FUNCTION_BLOCK Auto_rock
VAR_INPUT
	Safety_interlock:BOOL;
	Lh_depth:REAL;
	Rh_depth:REAL;
	Underground_despatch:BOOL;
	Right_brakes_on_dist:REAL;
	Left_brakes_on_dist:REAL;
	Tip_zone_up:REAL;
	Tip_zone_down:REAL;
	Box_zone_up:REAL;
	Box_zone_down:REAL;
	Rock_cycle_unlatch_dist:REAL;
	Loaded_skip_current:REAL;
END_VAR
VAR_OUTPUT
	Auto_ref:REAL;
	Starting_torque:REAL;
	Manual:BOOL;
	Auto:BOOL;
	Auto_go:BOOL;
	Auto_fwd:BOOL;
	Auto_rev:BOOL;
	Trail_brakes:BOOL;
	Fwd_incomplete:BOOL;
	Rev_incomplete:BOOL;
	Left_tip_zone:BOOL;
	Right_tip_zone:BOOL;
	Left_box_zone:BOOL;
	Right_box_zone:BOOL;
	Ready_to_load_rock:BOOL;
	Left_bank_zone:BOOL;
	Right_bank_zone:BOOL;
	ct_Skip_still_full:BOOL;
	ct_Auto_requirements:BOOL;
END_VAR
VAR_IN_OUT
	HMI_data:dut_Auto_rock;
	Levels:ARRAY[*] OF REAL;
END_VAR
VAR
	Auto_requirements_fault:BOOL;
	Rock_cycle_bypass_hmi:BOOL;
	Window_0: Window;
	Window_1: Window;
	R_TRIG_0: R_TRIG;
	R_TRIG_1: R_TRIG;
	TOF_0: TOF;
	F_TRIG_0: F_TRIG;
	BIT_TO_WORD_V0_0: BIT_TO_WORD_V0;
	WORD_TO_BIT_V0_0: WORD_TO_BIT_V0;
END_VAR

Zones();
Auto_mode();
Despatch();
Trail_brakes_m();
Auto_trips();
HMI_data_m();

METHOD Auto_mode
VAR_INPUT
END_VAR
VAR_INST // added by the converter: edge detectors and wires of the graphical bodies
    _w1, _w2 : BOOL;
    _w3 : ANY;
END_VAR
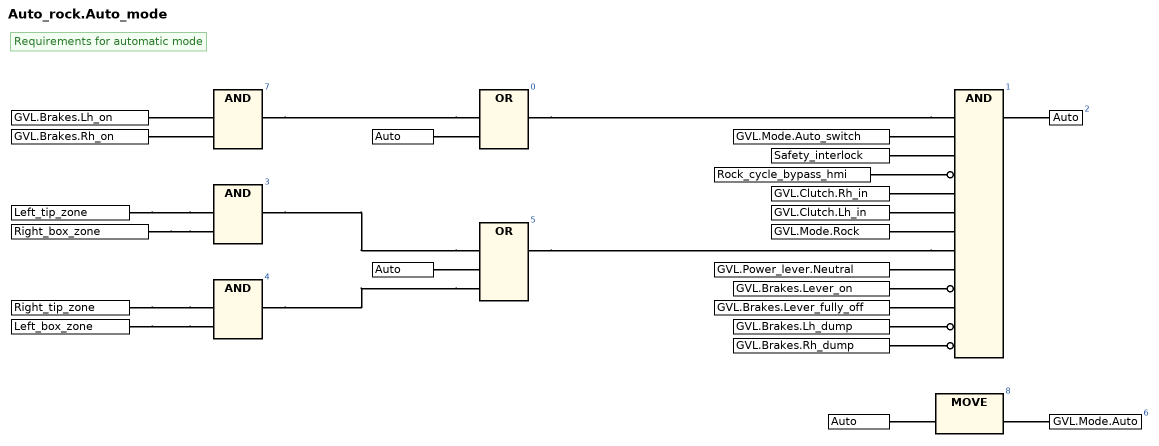
Auto := (_w1 OR Auto) AND GVL.Mode.Auto_switch AND Safety_interlock AND NOT Rock_cycle_bypass_hmi AND GVL.Clutch.Rh_in AND GVL.Clutch.Lh_in AND GVL.Mode.Rock AND _w2 AND GVL.Power_lever.Neutral AND NOT GVL.Brakes.Lever_on AND GVL.Brakes.Lever_fully_off AND NOT GVL.Brakes.Lh_dump AND NOT GVL.Brakes.Rh_dump;
_w2 := Left_tip_zone AND Right_box_zone OR Auto OR Right_tip_zone AND Left_box_zone;
GVL.Mode.Auto := _w3;
// Requirements for automatic mode
_w1 := GVL.Brakes.Lh_on AND GVL.Brakes.Rh_on;
_w3 := Auto;
END_METHOD

METHOD Auto_trips
VAR_INPUT
END_VAR
VAR_INST // added by the converter: edge detectors and wires of the graphical bodies
    _w1, _w2, _w3, _w4 : BOOL;
    _w5 : ANY;
END_VAR
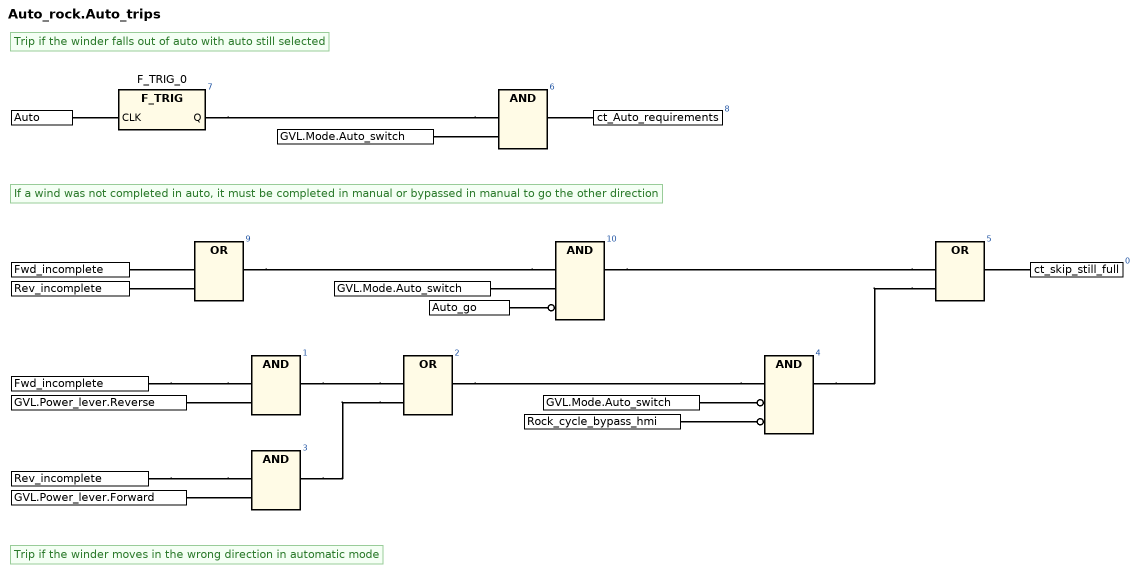
ct_skip_still_full := _w1;
_w3 := Fwd_incomplete AND GVL.Power_lever.Reverse OR _w2;
// Trip if the winder moves in the wrong direction in automatic mode
_w2 := Rev_incomplete AND GVL.Power_lever.Forward;
_w1 := _w4 OR _w3 AND NOT GVL.Mode.Auto_switch AND NOT Rock_cycle_bypass_hmi;
_w5 := F_TRIG_0.Q AND GVL.Mode.Auto_switch;
// Trip if the winder falls out of auto with auto still selected
F_TRIG_0(CLK := Auto); // F_TRIG
ct_Auto_requirements := _w5;
// If a wind was not completed in auto, it must be completed in manual or bypassed in manual to go the other direction
_w4 := (Fwd_incomplete OR Rev_incomplete) AND GVL.Mode.Auto_switch AND NOT Auto_go;
END_METHOD

METHOD Despatch
VAR_INPUT
END_VAR
VAR_INST // added by the converter: edge detectors and wires of the graphical bodies
    _w1, _w2, _w3, _w4, _w5, _w6, _w7, _w8, _w11, _w12, _w13 : BOOL;
    _w9, _w10 : REAL;
END_VAR
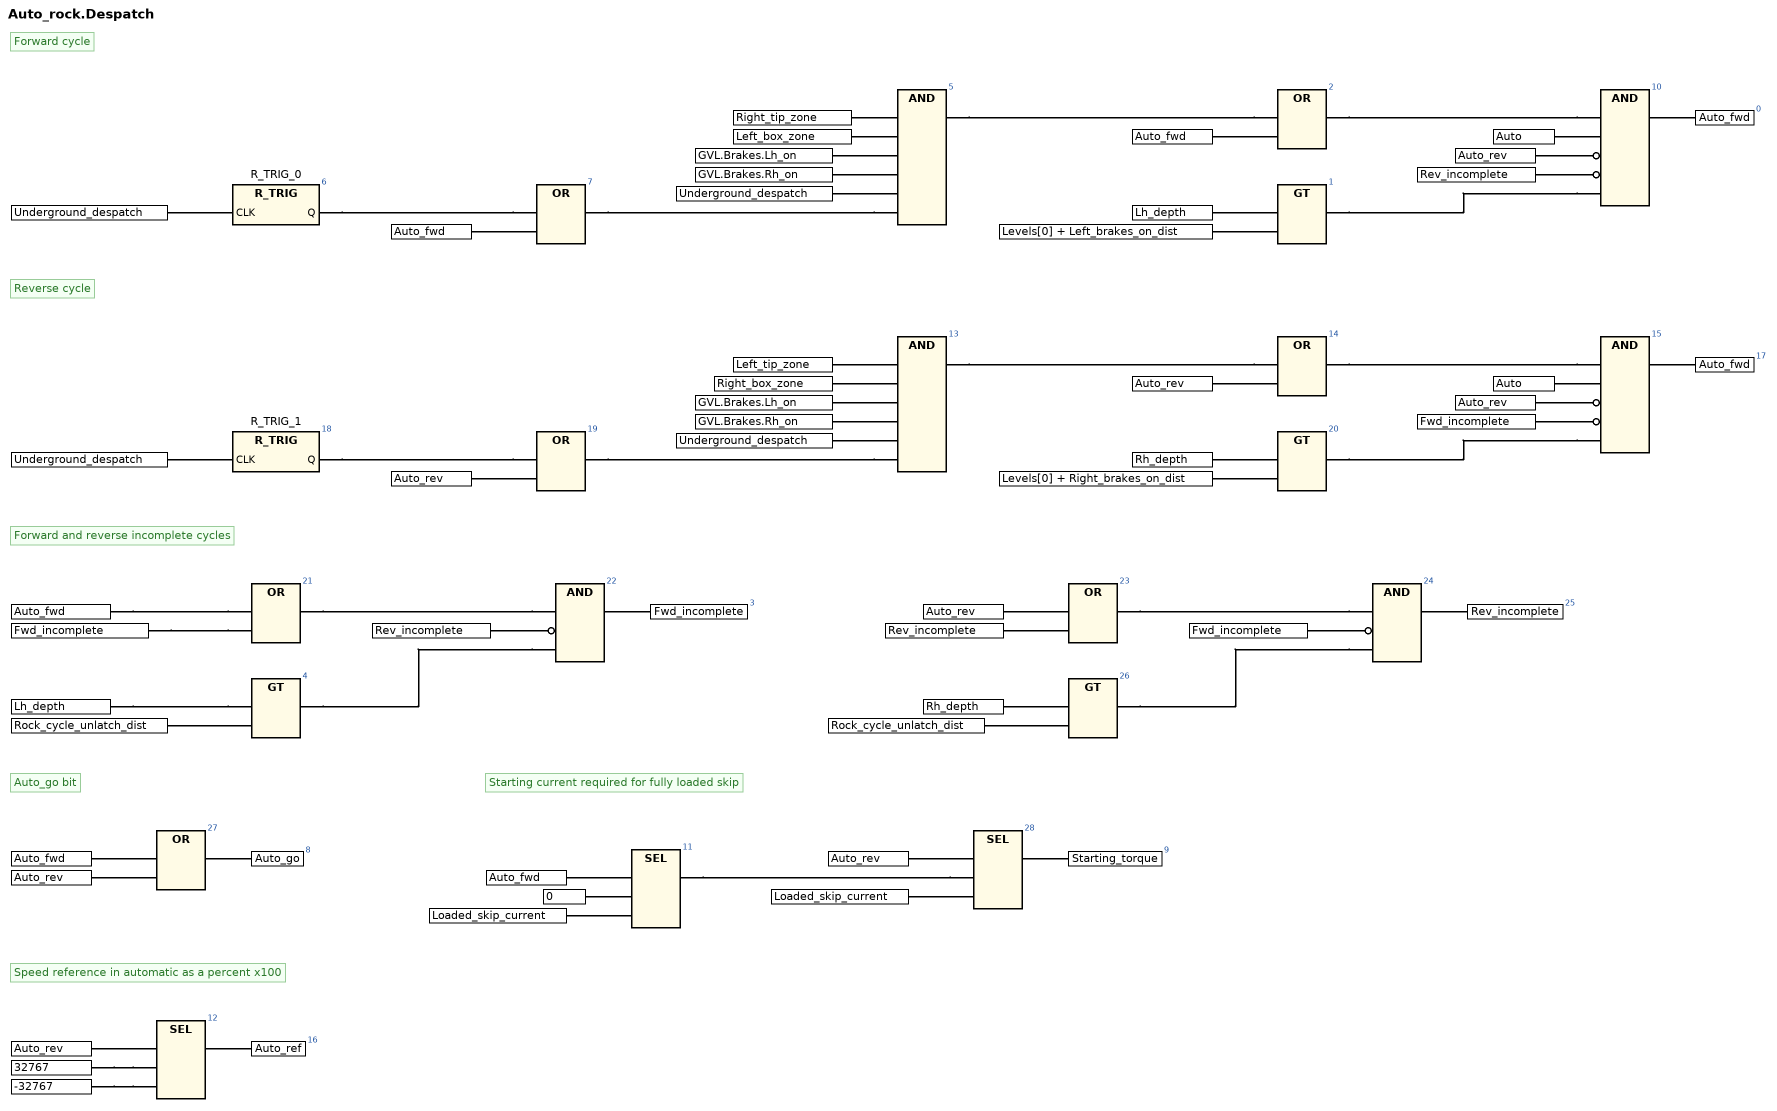
Auto_fwd := _w1;
_w2 := Lh_depth > (Levels[0] + Left_brakes_on_dist);
_w4 := _w3 OR Auto_fwd;
Fwd_incomplete := _w5;
_w6 := Lh_depth > Rock_cycle_unlatch_dist;
_w3 := Right_tip_zone AND Left_box_zone AND GVL.Brakes.Lh_on AND GVL.Brakes.Rh_on AND Underground_despatch AND _w7;
// Forward cycle
R_TRIG_0(CLK := Underground_despatch); // R_TRIG
_w7 := R_TRIG_0.Q OR Auto_fwd;
Auto_go := _w8;
Starting_torque := _w9;
_w1 := _w4 AND Auto AND NOT Auto_rev AND NOT Rev_incomplete AND _w2;
// Starting current required for fully loaded skip
_w10 := SEL(Auto_fwd, 0, Loaded_skip_current);
// Speed reference in automatic as a percent x100
Auto_ref := SEL(Auto_rev, 32767, -32767);
Auto_fwd := (Left_tip_zone AND Right_box_zone AND GVL.Brakes.Lh_on AND GVL.Brakes.Rh_on AND Underground_despatch AND _w11 OR Auto_rev) AND Auto AND NOT Auto_rev AND NOT Fwd_incomplete AND _w12;
// Reverse cycle
R_TRIG_1(CLK := Underground_despatch); // R_TRIG
_w11 := R_TRIG_1.Q OR Auto_rev;
_w12 := Rh_depth > (Levels[0] + Right_brakes_on_dist);
// Forward and reverse incomplete cycles
_w5 := (Auto_fwd OR Fwd_incomplete) AND NOT Rev_incomplete AND _w6;
Rev_incomplete := (Auto_rev OR Rev_incomplete) AND NOT Fwd_incomplete AND _w13;
_w13 := Rh_depth > Rock_cycle_unlatch_dist;
// Auto_go bit
_w8 := Auto_fwd OR Auto_rev;
_w9 := SEL(Auto_rev, _w10, Loaded_skip_current);
END_METHOD

METHOD HMI_data_m
VAR_INPUT
END_VAR
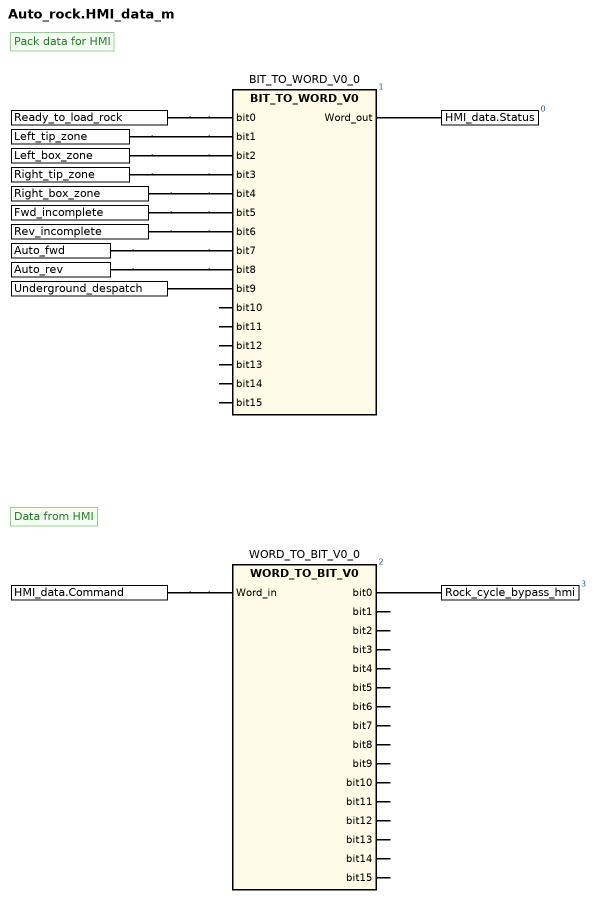
HMI_data.Status := BIT_TO_WORD_V0_0.Word_out;
// Pack data for HMI
BIT_TO_WORD_V0_0(
    bit0 := Ready_to_load_rock,
    bit1 := Left_tip_zone,
    bit2 := Left_box_zone,
    bit3 := Right_tip_zone,
    bit4 := Right_box_zone,
    bit5 := Fwd_incomplete,
    bit6 := Rev_incomplete,
    bit7 := Auto_fwd,
    bit8 := Auto_rev,
    bit9 := Underground_despatch); // BIT_TO_WORD_V0
// Data from HMI
WORD_TO_BIT_V0_0(Word_in := HMI_data.Command); // WORD_TO_BIT_V0
Rock_cycle_bypass_hmi := WORD_TO_BIT_V0_0.bit0;
END_METHOD

METHOD Trail_brakes_m
VAR_INPUT
END_VAR
VAR_INST // added by the converter: edge detectors and wires of the graphical bodies
    _w1, _w3 : BOOL;
    _w2 : ANY;
END_VAR
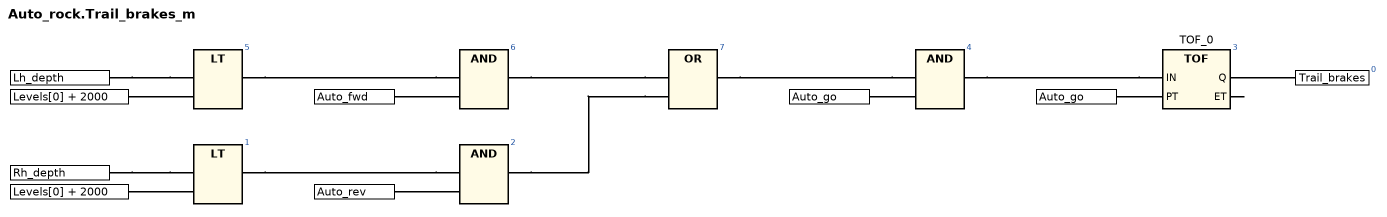
Trail_brakes := TOF_0.Q;
_w1 := Rh_depth < (Levels[0] + 2000) AND Auto_rev;
TOF_0(IN := _w2, PT := Auto_go); // TOF
_w2 := _w3 AND Auto_go;
_w3 := Lh_depth < (Levels[0] + 2000) AND Auto_fwd OR _w1;
END_METHOD

METHOD Zones
VAR_INPUT
END_VAR
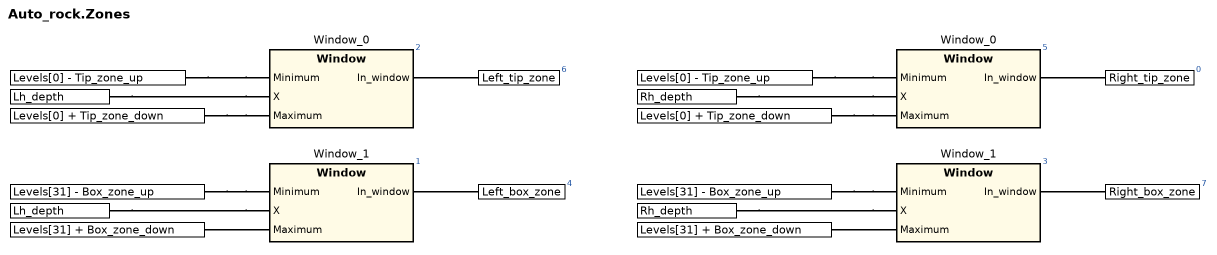
Right_tip_zone := Window_0.In_window;
Window_1(Minimum := Levels[31] - Box_zone_up, X := Lh_depth, Maximum := Levels[31] + Box_zone_down); // Window
Window_0(Minimum := Levels[0] - Tip_zone_up, X := Lh_depth, Maximum := Levels[0] + Tip_zone_down); // Window
Window_1(Minimum := Levels[31] - Box_zone_up, X := Rh_depth, Maximum := Levels[31] + Box_zone_down); // Window
Left_box_zone := Window_1.In_window;
Window_0(Minimum := Levels[0] - Tip_zone_up, X := Rh_depth, Maximum := Levels[0] + Tip_zone_down); // Window
Left_tip_zone := Window_0.In_window;
Right_box_zone := Window_1.In_window;
END_METHOD

END_FUNCTION_BLOCK

(* stored: Version 1.1.0.1, ProductVersion 3.1.4024.0
   POU Auto_rock: Id {4847b433-edf1-4a76-bd58-66bd69400c3d}, SpecialFunc None
   Method Auto_mode: Id {92b2812f-7f97-4d7e-9c77-d5cd38e31fe7}
   Method Auto_trips: Id {4fd9d4f2-6b65-4f13-8a68-c5d6e0bb2188}
   Method Despatch: Id {95aaba7e-b400-4252-84b4-e35cf08ca5aa}
   Method HMI_data_m: Id {6a5e0cc7-e463-4e2c-b4ec-30d5e3cc37e0}
   Method Trail_brakes_m: Id {72ee8853-6792-4147-9490-9c35f5b7bc74}
   Method Zones: Id {e9eb9c53-4772-45c5-8a1d-788c58e95169} *)
